// TIA Portal V20 export
FUNCTION "PreProcessing" : Void   // FC1, LAD
TITLE = PreProcessing
// V1.0  25.05.04  Test program by SG. Jeong
// stored: Namespace Safety, SetENOAutomatically false
BEGIN

REGION Network 1: Sending Acknowledge signal to BA010, ReelCut #1
   // Acknowledge signal transfer to  BA010, ReelCut #1
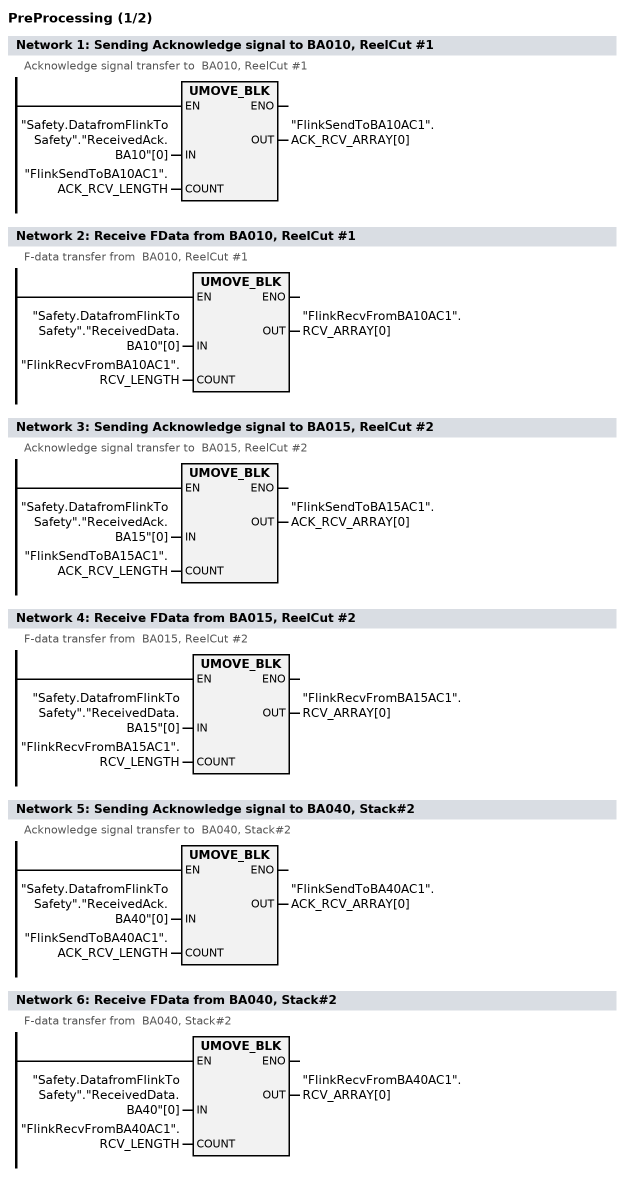
   UMOVE_BLK(IN := "Safety.DatafromFlinkToSafety"."ReceivedAck.BA10"[0],
             COUNT := "FlinkSendToBA10AC1".ACK_RCV_LENGTH,
             OUT => "FlinkSendToBA10AC1".ACK_RCV_ARRAY[0]);
END_REGION

REGION Network 2: Receive FData from BA010, ReelCut #1
   // F-data transfer from  BA010, ReelCut #1
   UMOVE_BLK(IN := "Safety.DatafromFlinkToSafety"."ReceivedData.BA10"[0],
             COUNT := "FlinkRecvFromBA10AC1".RCV_LENGTH,
             OUT => "FlinkRecvFromBA10AC1".RCV_ARRAY[0]);
END_REGION

REGION Network 3: Sending Acknowledge signal to BA015, ReelCut #2
   // Acknowledge signal transfer to  BA015, ReelCut #2
   UMOVE_BLK(IN := "Safety.DatafromFlinkToSafety"."ReceivedAck.BA15"[0],
             COUNT := "FlinkSendToBA15AC1".ACK_RCV_LENGTH,
             OUT => "FlinkSendToBA15AC1".ACK_RCV_ARRAY[0]);
END_REGION

REGION Network 4: Receive FData from BA015, ReelCut #2
   // F-data transfer from  BA015, ReelCut #2
   UMOVE_BLK(IN := "Safety.DatafromFlinkToSafety"."ReceivedData.BA15"[0],
             COUNT := "FlinkRecvFromBA15AC1".RCV_LENGTH,
             OUT => "FlinkRecvFromBA15AC1".RCV_ARRAY[0]);
END_REGION

REGION Network 5: Sending Acknowledge signal to BA040, Stack#2
   // Acknowledge signal transfer to  BA040, Stack#2
   UMOVE_BLK(IN := "Safety.DatafromFlinkToSafety"."ReceivedAck.BA40"[0],
             COUNT := "FlinkSendToBA40AC1".ACK_RCV_LENGTH,
             OUT => "FlinkSendToBA40AC1".ACK_RCV_ARRAY[0]);
END_REGION

REGION Network 6: Receive FData from BA040, Stack#2
   // F-data transfer from  BA040, Stack#2
   UMOVE_BLK(IN := "Safety.DatafromFlinkToSafety"."ReceivedData.BA40"[0],
             COUNT := "FlinkRecvFromBA40AC1".RCV_LENGTH,
             OUT => "FlinkRecvFromBA40AC1".RCV_ARRAY[0]);
END_REGION

REGION Network 7: Sending Acknowledge signal to BA060, Inspection
   // Acknowledge signal transfer to  BA060, Inspection
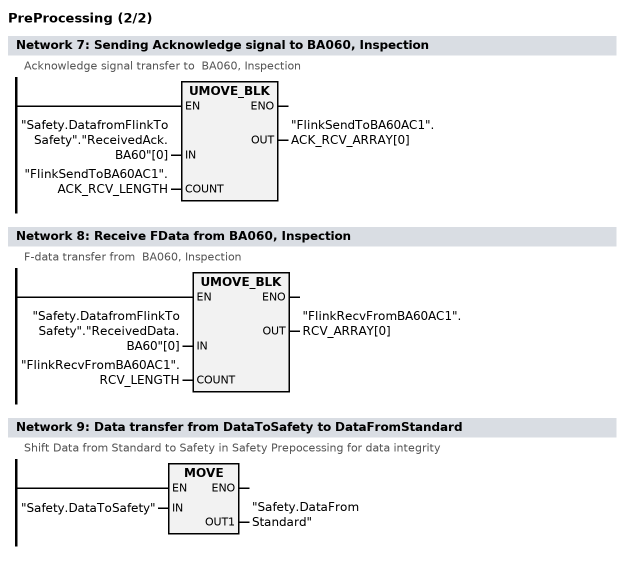
   UMOVE_BLK(IN := "Safety.DatafromFlinkToSafety"."ReceivedAck.BA60"[0],
             COUNT := "FlinkSendToBA60AC1".ACK_RCV_LENGTH,
             OUT => "FlinkSendToBA60AC1".ACK_RCV_ARRAY[0]);
END_REGION

REGION Network 8: Receive FData from BA060, Inspection
   // F-data transfer from  BA060, Inspection
   UMOVE_BLK(IN := "Safety.DatafromFlinkToSafety"."ReceivedData.BA60"[0],
             COUNT := "FlinkRecvFromBA60AC1".RCV_LENGTH,
             OUT => "FlinkRecvFromBA60AC1".RCV_ARRAY[0]);
END_REGION

REGION Network 9: Data transfer from DataToSafety to DataFromStandard
   // Shift Data from Standard to Safety in Safety Prepocessing for data integrity
   RUNG wire#powerrail
      Move(in := "Safety.DataToSafety", out1 => "Safety.DataFromStandard")
   END_RUNG
   // the same network as SCL:
   "Safety.DataFromStandard" := "Safety.DataToSafety";
END_REGION
END_FUNCTION
